Staubli VAL3: Control_List.pgx

public program Control_List(string& x_sItemName[], num& x_nSelectItem)
  local num l_nIndex
  local bool l_bRes
  local num l_nFrist
  local num l_nNum
  local bool l_bBlack
  local bool l_bBlank
  local num l_nCount
  local string l_sBuff
begin
  //说明：
  //函数功能：在划定的框内，把选中项给显示出来
  //l_nFirst  在列表中第一个显示的项的序号
  //x_nSelectItem  被选中的项的序号
  //l_nCount 合法列表项的项总数，如何数组中间为空，则可能被截断


  //1.参数初始化
  l_nFrist=0
  l_nCount=0

  //2.参数合法化判断，得到合法项的总数
  for l_nIndex=0 to size(x_sItemName)-1
    if x_sItemName[l_nIndex]==""
      l_nIndex=size(x_sItemName)
    else
      l_nCount=l_nCount+1
    endIf
  endFor

  //3.如果选中项大于列表长度
  x_nSelectItem=min(max(0,x_nSelectItem),l_nCount-1)
  if x_nSelectItem>=nPanelLengthY
    l_nFrist=x_nSelectItem-nPanelLengthY+1
  endIf


  //4.把列表给画出来
  for l_nIndex=0 to min(nPanelLengthY-1,l_nCount-l_nFrist-1)
    gotoxy(nPanelLTopX+1,nPanelLTopY+l_nIndex+1)
    setTextMode(sel(l_nIndex+l_nFrist==x_nSelectItem,1,0))
    //l_nNum=max(nPanelWidthX-getDisplayLen(x_sItemName[l_nIndex+l_nFrist])+len(x_sItemName[l_nIndex+l_nFrist]),nPanelWidthX)
   l_sBuff=left(x_sItemName[l_nIndex+l_nFrist]+"                                  ",nPanelWidthX)
   while getDisplayLen(l_sBuff)>nPanelWidthX
  l_sBuff=left(l_sBuff,len(l_sBuff)-1)
  endWhile
  put(l_sBuff)
//   left(x_sItemName[x_sItemName[l_nIndex+l_nFrist]],nPanelWidthX-)
//    put(left(x_sItemName[l_nIndex+l_nFrist]+"                            ",l_nNum))





  endFor


  //5.对剩下的进行补空
  setTextMode(0)
  while l_nIndex< nPanelLengthY
    gotoxy(nPanelLTopX+1,nPanelLTopY+l_nIndex+1)
    put(left("                               ",nPanelWidthX))
    l_nIndex=l_nIndex+1
  endWhile


end
